PROGRAM P001_Counter1
VAR
	count: INT;
END_VAR

count:=count+1;

END_PROGRAM

(* stored: Version 1.1.0.1, ProductVersion 3.1.4024.13
   POU P001_Counter1: Id {7d05dc1f-6454-42cd-b42b-390332ff6510}, SpecialFunc None *)
